TYPE TcoUr20_Inputs_v_1_x_x :
STRUCT
	Inputs AT %I* : ARRAY[0..63] OF BYTE;
END_STRUCT
END_TYPE

(* stored: Version 1.1.0.1, ProductVersion 3.1.4024.12
   DUT TcoUr20_Inputs_v_1_x_x: Id {26a40705-e58d-0fc2-3d98-35d604caf658} *)
